FUNCTION_BLOCK FloatArg IMPLEMENTS I_MutFloatArg
VAR
	_val			: LREAL;
END_VAR

PROPERTY Val : LREAL
GET
Val := _val;
END_GET
SET
_val := Val;
END_SET
END_PROPERTY

END_FUNCTION_BLOCK

(* stored: Version 1.1.0.1
   POU FloatArg: Id {00911996-c08a-42e6-b802-f28bf17d1565}, SpecialFunc None
   Property Val: Id {6d8da170-8112-482c-953b-21eacfd99080}
   Get Get: Id {d6a7f46b-4571-42d8-947d-f1572f1495d7}
   Set Set: Id {d2f51f5b-0ee9-40ab-898e-c4bd89ae55dc} *)
